PROGRAM MotionControl
VAR
END_VAR

END_PROGRAM

(* stored: Version 1.1.0.1, ProductVersion 3.1.4024.12
   POU MotionControl: Id {162d13a1-2db7-445d-83bf-25f4ef89db8f}, SpecialFunc None *)
